// TIA Portal V18 export
TYPE "UDT_DL_Vars"
// stored: IsFailsafeCompliant false
   STRUCT
      rOATtoHeatUpLine : Real;
      cReserve1 : Byte;
      cReserve2 : Byte;
      cDLPanelModeSelector : Byte := 16#3;
      rDayTankLevelAlarmMin : Array[1..2] of Real;
      rDayTankLevelStartFilling : Array[1..2] of Real;
      rDayTankLevelStopFilling : Array[1..2] of Real;
      rDayTankLevelAlarmMax : Array[1..2] of Real;
      cExericeSeconds : Array[1..2] of Byte;
      cMaxHoursWithoutRunToExerise : Array[1..2] of Byte;
      cActualHoursWithoutRunToExerise : Array[1..2] of Byte;
   END_STRUCT;
   // rDayTankLevelAlarmMin[1] := 50.0;
   // rDayTankLevelAlarmMin[2] := 51.0;
   // rDayTankLevelStartFilling[1] := 70.0;
   // rDayTankLevelStartFilling[2] := 71.0;
   // rDayTankLevelStopFilling[1] := 90.0;
   // rDayTankLevelStopFilling[2] := 91.1;
   // rDayTankLevelAlarmMax[1] := 95.0;
   // rDayTankLevelAlarmMax[2] := 96.0;
   // cExericeSeconds[1..2] := 16#FA;
   // cMaxHoursWithoutRunToExerise[1] := 16#A8;
   // cMaxHoursWithoutRunToExerise[2] := 16#A9;
END_TYPE
